TYPE ST_APP_STATE :
STRUCT
  AppInit             : E_PROGRESS;
  State            : E_INSTANCE_STATE;
END_STRUCT
END_TYPE

(* stored: Version 1.1.0.1, ProductVersion 3.1.4026.18
   DUT ST_APP_STATE: Id {0a63471f-5d7a-410d-84b1-8dfcda8dc179} *)
